//{attribute 'qualified_only'}
{attribute 'strict'}
TYPE eUniquenessMethos :
(
		PartCode 				:= 0 ,  //Machine ID and Partcode from Machine, Date and Time from PC
		PartCode_DateTime 		:= 1 ,  //Machine ID, Partcode,Date time from Machine. nothing from PC
		PartCode_LPC 			:= 2 ,  //Machine ID, Lifelong Production Count from Machine (9 Digit)
		WorkOrderNo_QtyCount	:= 3    //ERP WO Number with it's Qty count

);
END_TYPE

(* stored: Version 1.1.0.1, ProductVersion 3.1.4024.3
   EnumerationTextList eUniquenessMethos: Id {7108ee47-dee7-4a4c-87bf-3e260805d227} *)
